Omron CX-Programmer project NewProject (CX-Programmer 9.51)

# PLC my_first_project: CP1L L

## Global symbols (name address type ; comment)
W0.01 BOOL  ; comment

## Program NewProgram1 (cyclic task 0)
Local symbols
button_1 0.00 BOOL
button_2 0.01 BOOL  ; comment
button_3 0.02 BOOL  ; comment
out_1 100.00 BOOL  ; comment
out_2 100.01 BOOL  ; 3

### Section Section1

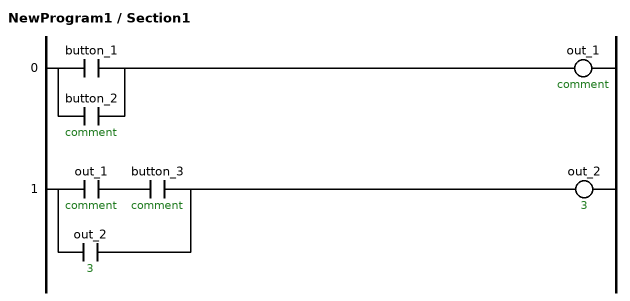
; rung 0
LD button_1
OR button_2  ; comment
OUT out_1  ; comment
; rung 1
LD out_1  ; comment
AND button_3  ; comment
OR out_2  ; 3
OUT out_2  ; 3

### Section END
; rung 0
END(001)